# EPICS substitutions: apps/bomApp/Db/bom_channels_sim.substitutions
file "db/bom_channel_sim.template" {
pattern { P R GAIN FLNK}
{ bom_sc_ai_ 0 20 0 }
{ bom_sc_ai_ 1 23 0 }
{ bom_sc_ai_ 2 21 0 }
{ bom_sc_ai_ 3 20 0 }
{ bom_sc_ai_ 4 21 0 }
{ bom_sc_ai_ 5 19 0 }
{ bom_sc_ai_ 6 17 0 }
{ bom_sc_ai_ 7 17 0 }
{ bom_sc_ai_ 8 20 0 }
{ bom_sc_ai_ 9 15 0 }
{ bom_sc_ai_ 10 15 0 }
{ bom_sc_ai_ 11 20 0 }
{ bom_sc_ai_ 12 23 0 }
{ bom_sc_ai_ 13 19 0 }
{ bom_sc_ai_ 14 19 0 }
{ bom_sc_ai_ 15 18 bom_sc_ai_sum_A.PROC }
}
